// TwinCAT 3 PLC project MAS418_PLC
// ProgramVersion: 3.1.4023.0
// libraries:
//   Tc2_Standard, * (Beckhoff Automation GmbH)
//   Tc2_System, * (Beckhoff Automation GmbH)
//   Tc3_Module, * (Beckhoff Automation GmbH)
// project tree:
//   / GlobalTextList.TcGTLO, PlcTask.TcTTO, Visualization Manager.TcVMO (not stored)
//   POUs/ MAIN.TcPOU
//   VISUs/ HMI.TcVIS
// real-time tasks:
//   TASK PlcTask: cycle T#10ms, priority 20, ADS port 350

CONFIGURATION MAS418_PLC
    RESOURCE PLC ON TwinCAT3
        TASK PlcTask(INTERVAL := T#10ms, PRIORITY := 20);
        PROGRAM MAIN WITH PlcTask : MAIN;
    END_RESOURCE
END_CONFIGURATION

// ---- POUs/MAIN.TcPOU
PROGRAM MAIN
VAR
	bEnable : BOOL := FALSE;
	bStart : BOOL := FALSE;
	nINT : INT := -32768;
	nUINT : UINT := 65535;
	fREAL : REAL := 255.255;
	sPowerStatus : STRING := 'Power Off';
	nFloatConversion : INT := 100; 
	fFloatConversion: LREAL :=10;
END_VAR

bEnable :=bStart;
fFloatConversion := INT_TO_REAL(nFloatConversion);

IF 
	bEnable
	THEN
	sPowerstatus := 'Power ON';
	ELSE
	sPowerStatus := 'Power OFF';	
END_IF

END_PROGRAM

// ---- GlobalTextList.TcGTLO
TEXTLIST GlobalTextList
  511 = '%iBOOL'
  607 = 'BOOL'
  896 = 'BOOL%i'
  806 = 'GroupBox'
  192 = 'INT'
  639 = 'INT%i'
  234 = 'REAL'
  772 = 'REAL%f'
  180 = 'REAL%i'
  40 = 'STRING'
  441 = 'STRING%s'
  152 = 'UINT'
  109 = 'UINT%i'
END_TEXTLIST

// ---- VISUs/HMI.TcVIS
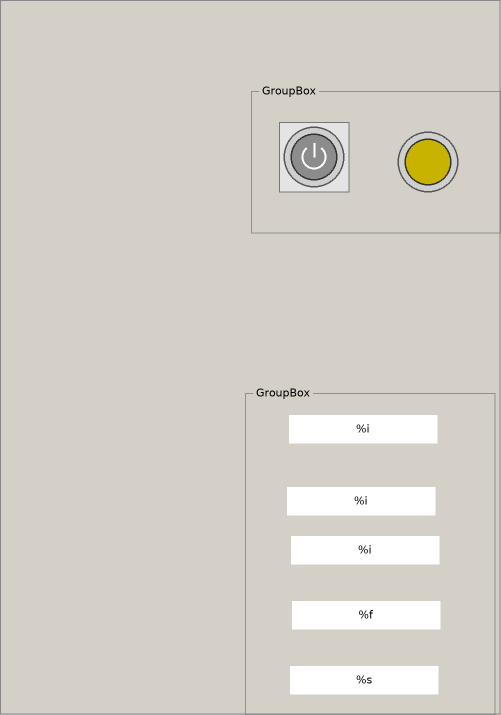
VISUALIZATION HMI  // 501x715
    GroupBox (251,83 250x150), "GroupBox"
        PowerSwitch (28,39 70x70), variable: MAIN.bStart, behaviour: TOGGLE, style: Switch-PowerSwitch-Gray
        Lamp1 (142,44 70x70), variable: MAIN.bStart, style: Lamp-Lamp1-Yellow
    GroupBox (245,385 250x330), "GroupBox"
        Textfield (45,150 150x30), "%i", text variable: MAIN.nUINT
        Textfield (46,215 150x30), "%f", text variable: MAIN.fREAL
        Textfield (43,29 150x30), "%i", text variable: Main.bEnable
        Textfield (44,280 150x30), "%s", text variable: MAIN.sPowerStatus
        Textfield (41,101 150x30), "%i", text variable: MAIN.nINT
END_VISUALIZATION
